FUNCTION_BLOCK FB_LoadCell_Smowo EXTENDS FB_ModbusSlaveRtu IMPLEMENTS I_Weight
VAR
	lrValueRaw : LREAL;
	lrValueGram : LREAL;
	lrValueKg : LREAL;
	TmpData : U_Word2Dint;
	bEnableReallyError : BOOL;
	lrRawValue : LREAL; // receive from module
	lrTareValue : LREAL; // Value at tare
END_VAR

tonConfirmReallyError(
	IN := bModbusError,
	PT := timeConfirmReallyError,
	Q => bReallyError 
);
SUPER^();

METHOD Convert : BOOL
VAR_INPUT
	iRegionNo	: 	INT;
	pReadData	:	POINTER TO word;
END_VAR
CASE iRegionNo OF
	0:
		TmpData.iWord[1] := pReadData[0];
		TmpData.iWord[0] := pReadData[1];
		lrRawValue := DINT_TO_LREAL(TmpData.idInt);
		lrValueGram :=  lrRawValue-lrTareValue;
		lrValueKg := lrValueGram * 0.001;
END_CASE
END_METHOD

PROPERTY EnableReallyError : bool
GET
EnableReallyError := bEnableReallyError;
END_GET
SET
bEnableReallyError := EnableReallyError;
END_SET
END_PROPERTY

METHOD FirstCycle // must be call once time 
VAR_INPUT
	sName : STRING;
	iUnitID : BYTE ; // modbus address of the device : 1- 255
END_VAR
THIS^.sName := sName;
THIS^.iUnitID := iUnitID;

arrAddressRead[0][0] := 0;
arrAddressRead[0][1] := 2;
arrAddressRead[0][2] := TC_ModbusBase.E_ModbusFunction.ReadHoldingRegisters;
iNumAddRegionRead := 1;
END_METHOD

PROPERTY TareValue : Lreal
GET
TareValue := lrTareValue;
END_GET
SET
lrTareValue := TareValue;
END_SET
END_PROPERTY

PROPERTY ValueGram : reference to lreal
GET
ValueGram REF= lrValueGram;
END_GET
END_PROPERTY

PROPERTY ValueKg : reference to lreal
GET
ValueKg ref= lrValueKg;
END_GET
END_PROPERTY

END_FUNCTION_BLOCK

(* stored: Version 1.1.0.1, ProductVersion 3.1.4024.12
   POU FB_LoadCell_Smowo: Id {4658126e-c473-4426-805d-4ba545f65734}, SpecialFunc None
   Method Convert: Id {f612aa90-cf6b-4e46-acd4-79a4601d15a3}
   Property EnableReallyError: Id {2decdeb6-2b10-4472-9b77-4051f7655889}
   Get Get: Id {8549703a-5b10-49ec-994b-e05383b23b6c}
   Set Set: Id {ac143162-8e09-46fe-98c2-849cc191349a}
   Method FirstCycle: Id {21c18c7d-3744-4286-a670-437cfb3ae6c5}
   Property TareValue: Id {4d479054-a0dc-41b6-ab08-8f7d7fb120b6}
   Get Get: Id {24ca55aa-d932-4a57-9fb3-e7f7e29ecd84}
   Set Set: Id {6e40eb58-4f9e-4e2a-8057-6f661f32b8f8}
   Property ValueGram: Id {6bfa4383-7f76-4f9d-aa73-cd9028500bbe}
   Get Get: Id {d057e907-b377-4627-a8a5-ae196526c980}
   Property ValueKg: Id {bc5da4ff-2b2d-45e3-8907-6cce7b8feed0}
   Get Get: Id {c7faa42d-f77d-4337-9619-3980a6132df5} *)
